FUNCTION_BLOCK TEST_EQN (* Test EQ functions of numerical values *)
  (* Standard: IEC 61499-1 *)
  (* Version 0.0, 2006-09-11, JHC, Holobloc Inc *)
  (* Compiler header: package fb.rt.test; *)
  (* Compiler classdef: SimpleFB *)
  (* Compiler Java Sun JDK 1.5.0 *)
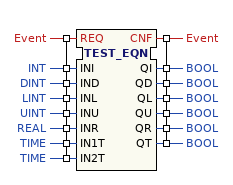
  EVENT_INPUT
    REQ WITH INI, INL, INU, IND, INR, IN1T, IN2T;
  END_EVENT
  EVENT_OUTPUT
    CNF WITH QI, QD, QL, QU, QR, QT;
  END_EVENT
  VAR_INPUT
    INI : INT;
    IND : DINT;
    INL : LINT;
    INU : UINT;
    INR : REAL;
    IN1T : TIME;
    IN2T : TIME;
  END_VAR
  VAR_OUTPUT
    QI : BOOL;
    QD : BOOL;
    QL : BOOL;
    QU : BOOL;
    QR : BOOL;
    QT : BOOL;
  END_VAR
  ALGORITHM REQ IN FBD:
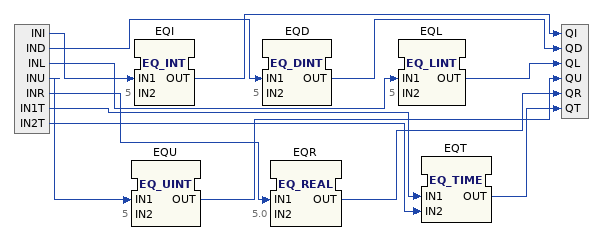
    FBS
      EQI : EQ_INT(IN2 := 5);
      EQD : EQ_DINT(IN2 := 5);
      EQL : EQ_LINT(IN2 := 5);
      EQU : EQ_UINT(IN2 := 5);
      EQR : EQ_REAL(IN2 := 5.0);
      EQT : EQ_TIME;
    END_FBS
    DATA_CONNECTIONS
      INI TO EQI.IN1;
      IND TO EQD.IN1;
      INL TO EQL.IN1;
      INU TO EQU.IN1;
      INR TO EQR.IN1;
      EQI.OUT TO QI;
      EQD.OUT TO QD;
      EQL.OUT TO QL;
      EQU.OUT TO QU;
      EQR.OUT TO QR;
      EQT.OUT TO QT;
      IN1T TO EQT.IN1;
      IN2T TO EQT.IN2;
    END_CONNECTIONS
  END_ALGORITHM
END_FUNCTION_BLOCK
